{attribute 'qualified_only'}
{attribute 'strict'}
{attribute 'to_string'}
TYPE E_Modes :
(
	Automatic 		:= 0,
	NonAutomatic 	:= 1,
	Manual			:= 2
);
END_TYPE

(* stored: Version 1.1.0.1, ProductVersion 3.1.4026.18
   DUT E_Modes: Id {7d069958-7972-4944-9884-6ee9d67b58d6} *)
